// TIA Portal project "osnovni projekt" (V17)
// Neki, neki, bla bla bla

(* hardware
DEVICE "S7-300/ET200M station_1"  S7-300 station
   slot 0: "Rail_0"  Rail  6ES7 390-1***0-0AA0
   slot 1: "PS 307 5A_1"  PS 307 5A  6ES7 307-1EA00-0AA0
   slot 2: "PLC_1"  CPU 315F-2 PN/DP  6ES7 315-2FJ14-0AB0  V3.2
      slot 2: "PROFINET interface_1"  PN-IO
         slot 1: "Port_1"  Port
         slot 2: "Port_2"  Port
   slot 4: "DI 16/DO 16x24VDC/0.5A_1"  DI16/DO16 x 24V / 0.5A  6ES7 323-1BL00-0AA0
   slot 5: "AI 4/AO 2x8BIT_1"  AI4/AO2 x 8 bits  6ES7 334-0CE01-0AA0
*)

// ===== PLC "PLC_1"  CPU 315F-2 PN/DP =====

DATA_BLOCK "Main_Safety_RTG1_DB"   // DB1, F_DB
{ S7_Optimized_Access := 'FALSE' }
VERSION : 0.1
// stored: InstanceOfName Main_Safety_RTG1
"Main_Safety_RTG1"
BEGIN
END_DATA_BLOCK

DATA_BLOCK "Data_block_1"   // DB4
{ S7_Optimized_Access := 'FALSE' }
VERSION : 0.1
   VAR
      Ventil1 : Bool;
      Ventil2 : Bool;
      Ventil3 : Bool;
      Ventil4 : Bool;
      Ventil5 : Bool;
      Crpalka : Int;
      Rezervoar : Int;
      hisica1 : Int;
      hisica2 : Int;
      hisica3 : Int;
      hisica4 : Int;
      hisica5 : Int;
   END_VAR
BEGIN
END_DATA_BLOCK

FUNCTION_BLOCK "Main_Safety_RTG1"   // FB1, F_LAD
{ S7_Optimized_Access := 'FALSE' }
BEGIN
END_FUNCTION_BLOCK

FUNCTION_BLOCK "Vsota pretoka na glavnem ventilu"   // FB10, SCL
{ S7_Optimized_Access := 'FALSE' }
VERSION : 0.1
   VAR_INPUT
      V1 : Bool;
      V2 : Bool;
      V3 : Bool;
      V4 : Bool;
      V5 : Bool;
   END_VAR
   VAR_OUTPUT
      Pretok : Int;
   END_VAR
BEGIN
   IF _condition_ THEN
       // Statement section IF
       ;
   END_IF;
END_FUNCTION_BLOCK

ORGANIZATION_BLOCK "Main"   // OB1, FBD
TITLE = "Main Program Sweep (Cycle)"
{ S7_Optimized_Access := 'FALSE' }
VERSION : 0.1
   VAR_TEMP
      OB1_EV_CLASS : Byte;   // Bits 0-3 = 1 (Coming event), Bits 4-7 = 1 (Event class 1)
      OB1_SCAN_1 : Byte;   // 1 (Cold restart scan 1 of OB 1), 3 (Scan 2-n of OB 1)
      OB1_PRIORITY : Byte;   // Priority of OB Execution
      OB1_OB_NUMBR : Byte;   // 1 (Organization block 1, OB1)
      OB1_RESERVED_1 : Byte;   // Reserved for system
      OB1_RESERVED_2 : Byte;   // Reserved for system
      OB1_PREV_CYCLE : Int;   // Cycle time of previous OB1 scan (milliseconds)
      OB1_MIN_CYCLE : Int;   // Minimum cycle time of OB1 (milliseconds)
      OB1_MAX_CYCLE : Int;   // Maximum cycle time of OB1 (milliseconds)
      OB1_DATE_TIME : Date_And_Time;   // Date and time OB1 started
   END_VAR
BEGIN

REGION Network 1
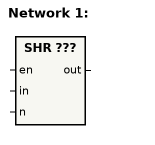
   <??.?> := SHR();
END_REGION
END_ORGANIZATION_BLOCK

ORGANIZATION_BLOCK "CYC_INT5_RTG1"   // OB35, LAD
TITLE = "Cyclic Interrupt"
{ S7_Optimized_Access := 'FALSE' }
VERSION : 0.1
   VAR_TEMP
      OB35_EV_CLASS : Byte;   // Bits 0-3 = 1 (Coming event), Bits 4-7 = 1 (Event class 1)
      OB35_STRT_INF : Byte;   // 16#36 (OB 35 has started)
      OB35_PRIORITY : Byte;   // Priority of OB Execution
      OB35_OB_NUMBR : Byte;   // 35 (Organization block 35, OB35)
      OB35_RESERVED_1 : Byte;   // Reserved for system
      OB35_RESERVED_2 : Byte;   // Reserved for system
      OB35_PHASE_OFFSET : Word;   // Phase offset (msec)
      OB35_RESERVED_3 : Int;   // Reserved for system
      OB35_EXC_FREQ : Int;   // Frequency of execution (msec)
      OB35_DATE_TIME : Date_And_Time;   // Date and time OB35 started
   END_VAR
BEGIN

REGION Network 1
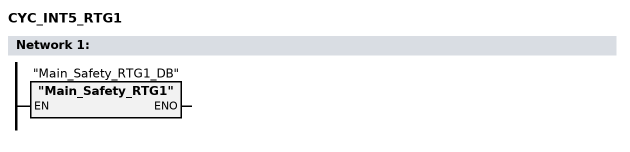
   RUNG wire#powerrail
      "Main_Safety_RTG1_DB"()
   END_RUNG
   // the same network as SCL:
   "Main_Safety_RTG1_DB"();   // "Main_Safety_RTG1"
END_REGION
END_ORGANIZATION_BLOCK